{attribute 'qualified_only'}
{attribute 'strict'}
TYPE status :
(START,
LEVELCHECK,
FILL,
HEAT,
HEATING,
BREW,
WATERREADY,
INTENSITY,
SUGAR,
READY,
CLEAN,
END,
OldState
) := START;
END_TYPE

(* stored: Version 1.1.0.1, ProductVersion 3.1.4024.15
   DUT status: Id {1a3340a8-f4e3-4153-85dc-b8d423a4a911} *)
